INTERFACE ITF_SaMElement EXTENDS ITF_BaseComponent

METHOD PUBLIC InvokeStateForTopElement : BOOL
VAR_INPUT
	itfTopElement		: ITF_BaseSaMStateMethod;
END_VAR
END_METHOD

METHOD PUBLIC IsActive : BOOL
VAR_INPUT
END_VAR
END_METHOD

(*			
	EVERDE sp. z o.o.
	Rafał Osajda		03.11.2025		TC 4024.66
	Zwraca czy element jest właczony w systemie
*)
METHOD PUBLIC IsEnabled : BOOL
VAR_INPUT
END_VAR
END_METHOD

METHOD PUBLIC ResetTime
VAR_INPUT
END_VAR
END_METHOD

(*			
	EVERDE sp. z o.o.
	Rafał Osajda		03.11.2025		TC 4024.66
	Ustawia czy dane element jest aktywny
*)
METHOD PUBLIC SetActive
VAR_INPUT
	bIN			: BOOL;
END_VAR
END_METHOD

(*			
	EVERDE sp. z o.o.
	Rafał Osajda		03.11.2025		TC 4024.66
	Ustawie czy element jest włączony w systemie
*)
METHOD PUBLIC SetEnabled
VAR_INPUT
	bIN			: BOOL;
END_VAR
END_METHOD

END_INTERFACE

(* stored: Version 1.1.0.1
   Itf ITF_SaMElement: Id {18e351e5-c377-09bd-199b-8ece74b821e4}
   Method InvokeStateForTopElement: Id {0f361f4f-cbec-0bac-0fc7-5725dafc2c84}
   Method IsActive: Id {c8d946d6-c2d5-0d48-0aaf-5a6a7c6a5209}
   Method IsEnabled: Id {ba56d189-2af0-0454-102a-8d822d334396}
   Method ResetTime: Id {52be7068-663a-05b0-36be-1a659653294f}
   Method SetActive: Id {8ae1fb1b-a80b-0a21-01d7-3a0d8be2ef76}
   Method SetEnabled: Id {ba2fccb0-69d6-0227-3d03-d59fb2553566} *)
